TYPE ST_StaticOutput :
STRUCT
    Output          :INT;
    State           :BYTE;
END_STRUCT
END_TYPE

(* stored: Version 1.1.0.1, ProductVersion 3.1.4024.9
   DUT ST_StaticOutput: Id {a0700f2a-4726-4cef-9ebd-ff78dade332d} *)
